FUNCTION_BLOCK FB_TimeSwitch_V2
VAR_INPUT
	b_Enable: BOOL;
	b_StatusOn: BOOL;
	structSystemTime: timestruct;
	byte_MoFr_Open_Hour: BYTE;
	byte_MoFr_Open_Minute: BYTE;
	byte_MoFr_Close_Hour: BYTE;
	byte_MoFr_Close_Minute: BYTE;
	byte_Sa_Open_Hour: BYTE;
	byte_Sa_Open_Minute: BYTE;
	byte_Sa_Close_Hour: BYTE;
	byte_Sa_Close_Minute: BYTE;	
	byte_So_Open_Hour: BYTE;
	byte_So_Open_Minute: BYTE;
	byte_So_Close_Hour: BYTE;
	byte_So_Close_Minute: BYTE;
	real_Offset_Start: REAL;
	real_Offset_Stop: REAL;	
	b_On_Manual: BOOL;
	b_Off_Manual: BOOL;
END_VAR
VAR_OUTPUT
	b_Output_On: BOOL;
	b_Error: BOOL;
END_VAR
VAR
	TON_0: ton;
	byte_Day :BYTE;		// 0: Sunday, 1: Monday,....
	time_now             		: TIME;
	time_MoFr_Open             	: TIME;
	time_MoFr_Close             : TIME;
	time_Sa_Open             	: TIME;
	time_Sa_Close             	: TIME;
	time_So_Open             	: TIME;
	time_So_Close             	: TIME;
	

	RS_0: rs;
	R_TRIG_0: r_trig;
	R_TRIG_1: r_trig;
	dt_Test: DATE_AND_TIME;
	tod_test: TIME_OF_DAY;
	time_temp: TIME;
	time_Start_MoFr_Calc: TIME;
	time_Stop_MoFr_Calc: TIME;
	time_Start_Sa_Calc: TIME;
	time_Stop_Sa_Calc: TIME;
	time_Start_So_Calc: TIME;
	time_Stop_So_Calc: TIME;
	
	FB_WeeklyTimeSwitch_MoFr: FB_WeeklyTimeSwitch;
	FB_WeeklyTimeSwitch_Sa: FB_WeeklyTimeSwitch;
	FB_WeeklyTimeSwitch_So: FB_WeeklyTimeSwitch;
	RS_manu: rs;
	b_Auto_on: BOOL;

	R_TRIG_2: r_trig;
	R_TRIG_3: r_trig;
	F_TRIG_0: f_trig;
	R_TRIG_4: r_trig;
	R_TRIG_FirstCycle: r_trig;
	time_Zero             	: TIME;
	
END_VAR
VAR // added by the converter: edge detectors and wires of the graphical bodies
    _w1 : DATE_AND_TIME;
    _w2 : TIME_OF_DAY;
    _w3 : BOOL;
END_VAR

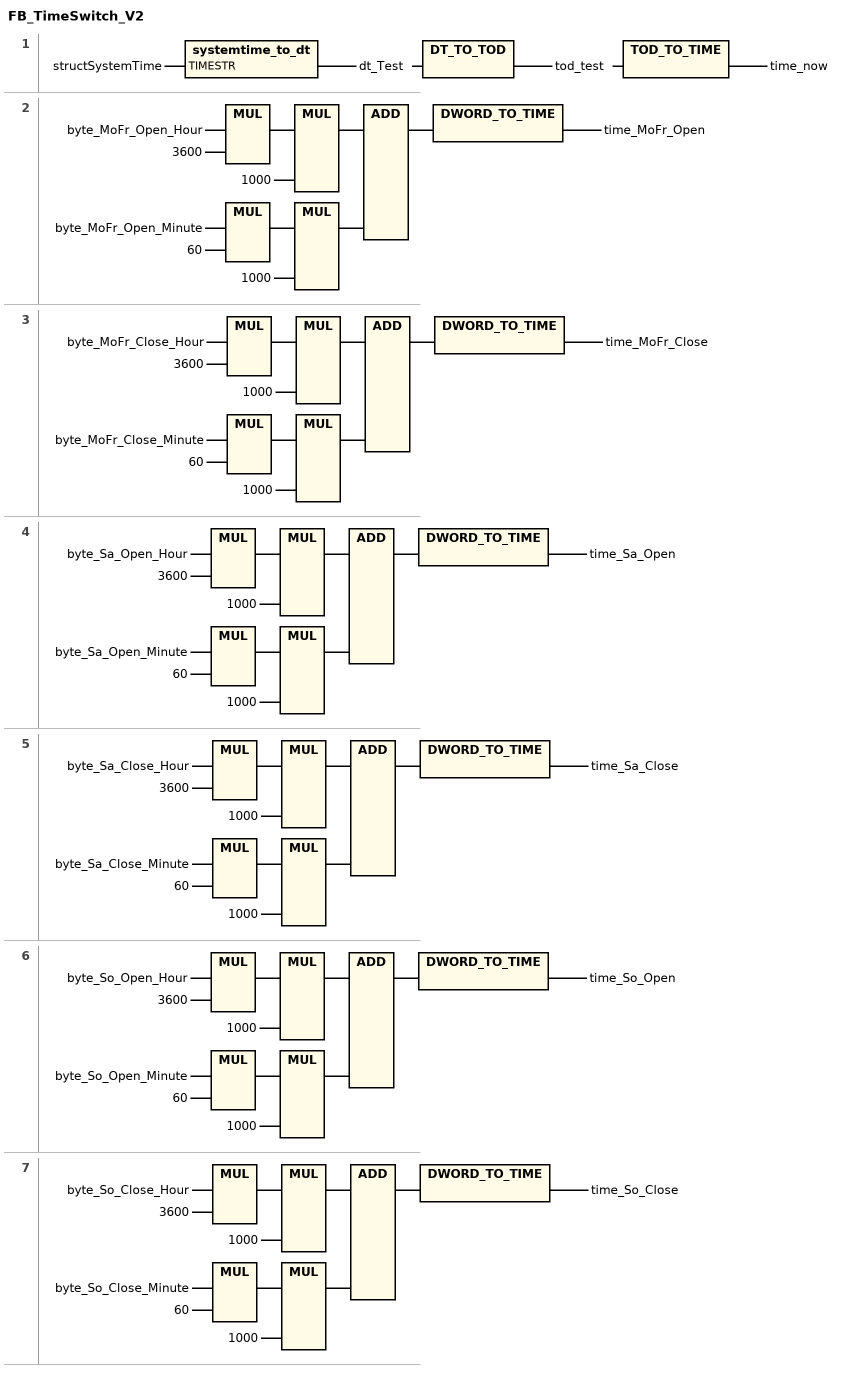
// NETWORK 1
_w1 := systemtime_to_dt(TIMESTR := structSystemTime);
dt_Test := _w1;
_w2 := DT_TO_TOD(_w1);
tod_test := _w2;
time_now := TOD_TO_TIME(_w2);

// NETWORK 2
time_MoFr_Open := DWORD_TO_TIME((byte_MoFr_Open_Hour * 3600) * 1000 + (byte_MoFr_Open_Minute * 60) * 1000);

// NETWORK 3
time_MoFr_Close := DWORD_TO_TIME((byte_MoFr_Close_Hour * 3600) * 1000 + (byte_MoFr_Close_Minute * 60) * 1000);

// NETWORK 4
time_Sa_Open := DWORD_TO_TIME((byte_Sa_Open_Hour * 3600) * 1000 + (byte_Sa_Open_Minute * 60) * 1000);

// NETWORK 5
time_Sa_Close := DWORD_TO_TIME((byte_Sa_Close_Hour * 3600) * 1000 + (byte_Sa_Close_Minute * 60) * 1000);

// NETWORK 6
time_So_Open := DWORD_TO_TIME((byte_So_Open_Hour * 3600) * 1000 + (byte_So_Open_Minute * 60) * 1000);

// NETWORK 7
time_So_Close := DWORD_TO_TIME((byte_So_Close_Hour * 3600) * 1000 + (byte_So_Close_Minute * 60) * 1000);

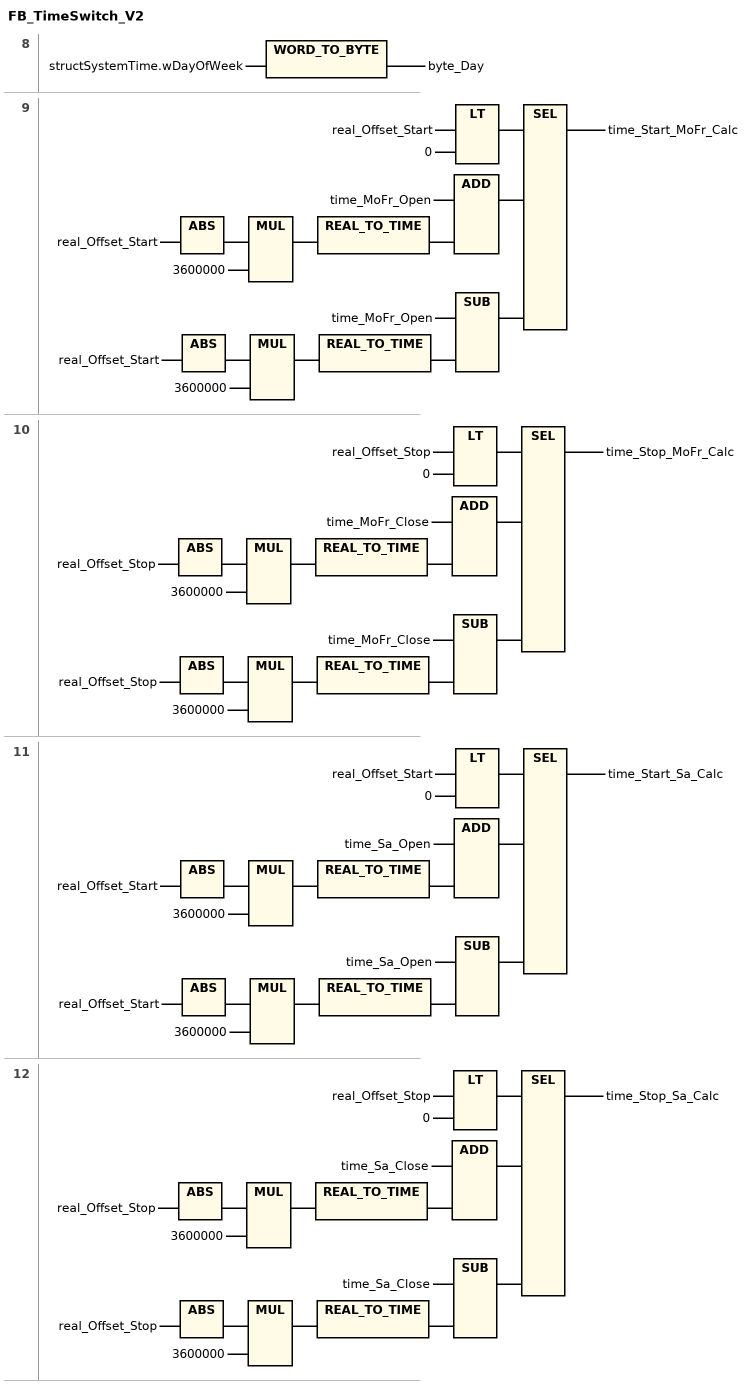
// NETWORK 8
byte_Day := WORD_TO_BYTE(structSystemTime.wDayOfWeek);

// NETWORK 9
time_Start_MoFr_Calc := SEL(real_Offset_Start < 0, time_MoFr_Open + REAL_TO_TIME(ABS(real_Offset_Start) * 3600000), time_MoFr_Open - REAL_TO_TIME(ABS(real_Offset_Start) * 3600000));

// NETWORK 10
time_Stop_MoFr_Calc := SEL(real_Offset_Stop < 0, time_MoFr_Close + REAL_TO_TIME(ABS(real_Offset_Stop) * 3600000), time_MoFr_Close - REAL_TO_TIME(ABS(real_Offset_Stop) * 3600000));

// NETWORK 11
time_Start_Sa_Calc := SEL(real_Offset_Start < 0, time_Sa_Open + REAL_TO_TIME(ABS(real_Offset_Start) * 3600000), time_Sa_Open - REAL_TO_TIME(ABS(real_Offset_Start) * 3600000));

// NETWORK 12
time_Stop_Sa_Calc := SEL(real_Offset_Stop < 0, time_Sa_Close + REAL_TO_TIME(ABS(real_Offset_Stop) * 3600000), time_Sa_Close - REAL_TO_TIME(ABS(real_Offset_Stop) * 3600000));

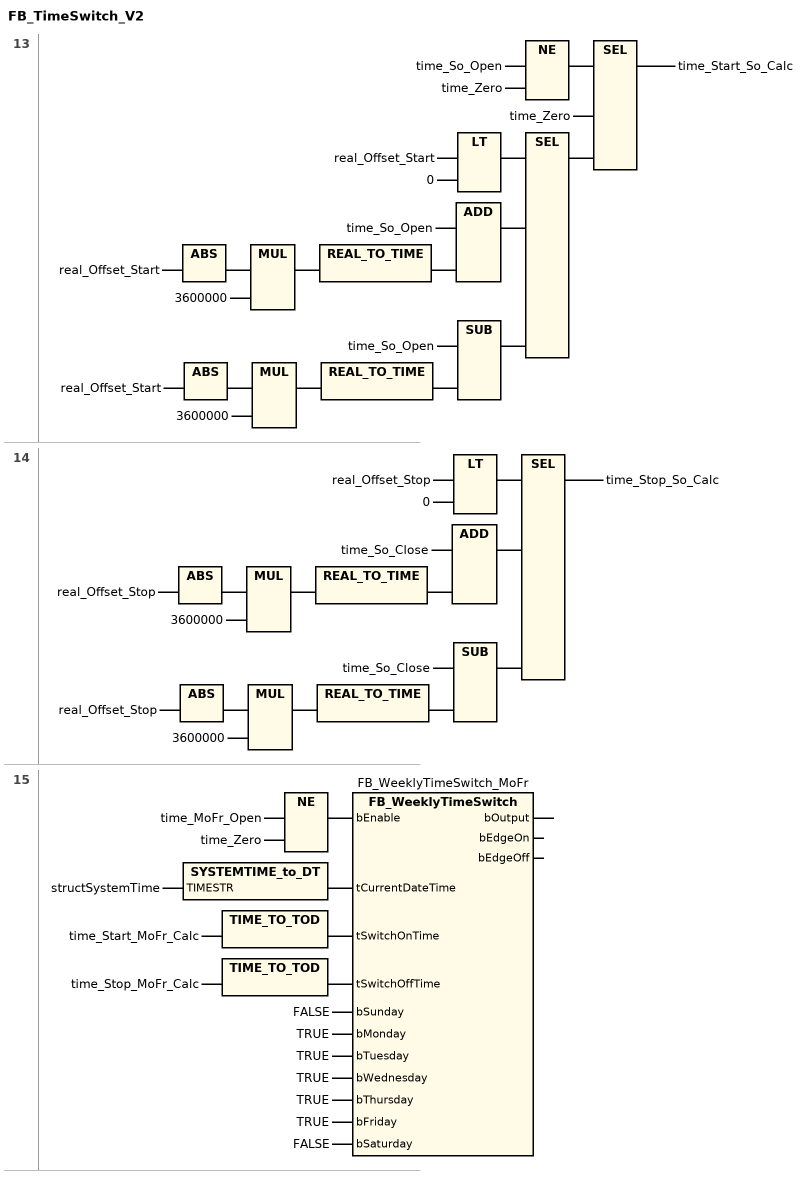
// NETWORK 13
time_Start_So_Calc := SEL(time_So_Open <> time_Zero, time_Zero, SEL(real_Offset_Start < 0, time_So_Open + REAL_TO_TIME(ABS(real_Offset_Start) * 3600000), time_So_Open - REAL_TO_TIME(ABS(real_Offset_Start) * 3600000)));

// NETWORK 14
time_Stop_So_Calc := SEL(real_Offset_Stop < 0, time_So_Close + REAL_TO_TIME(ABS(real_Offset_Stop) * 3600000), time_So_Close - REAL_TO_TIME(ABS(real_Offset_Stop) * 3600000));

// NETWORK 15
FB_WeeklyTimeSwitch_MoFr(
    bEnable := time_MoFr_Open <> time_Zero,
    tCurrentDateTime := SYSTEMTIME_to_DT(TIMESTR := structSystemTime),
    tSwitchOnTime := TIME_TO_TOD(time_Start_MoFr_Calc),
    tSwitchOffTime := TIME_TO_TOD(time_Stop_MoFr_Calc),
    bSunday := FALSE,
    bMonday := TRUE,
    bTuesday := TRUE,
    bWednesday := TRUE,
    bThursday := TRUE,
    bFriday := TRUE,
    bSaturday := FALSE); // FB_WeeklyTimeSwitch

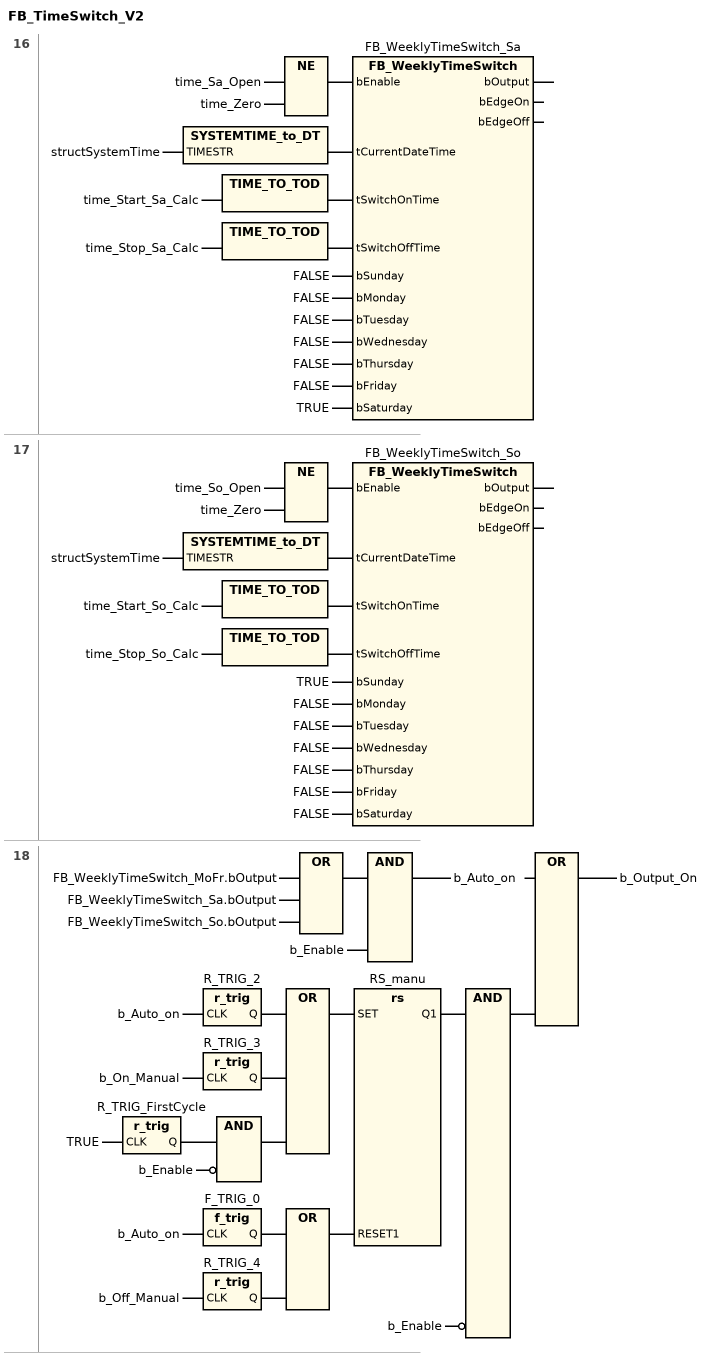
// NETWORK 16
FB_WeeklyTimeSwitch_Sa(
    bEnable := time_Sa_Open <> time_Zero,
    tCurrentDateTime := SYSTEMTIME_to_DT(TIMESTR := structSystemTime),
    tSwitchOnTime := TIME_TO_TOD(time_Start_Sa_Calc),
    tSwitchOffTime := TIME_TO_TOD(time_Stop_Sa_Calc),
    bSunday := FALSE,
    bMonday := FALSE,
    bTuesday := FALSE,
    bWednesday := FALSE,
    bThursday := FALSE,
    bFriday := FALSE,
    bSaturday := TRUE); // FB_WeeklyTimeSwitch

// NETWORK 17
FB_WeeklyTimeSwitch_So(
    bEnable := time_So_Open <> time_Zero,
    tCurrentDateTime := SYSTEMTIME_to_DT(TIMESTR := structSystemTime),
    tSwitchOnTime := TIME_TO_TOD(time_Start_So_Calc),
    tSwitchOffTime := TIME_TO_TOD(time_Stop_So_Calc),
    bSunday := TRUE,
    bMonday := FALSE,
    bTuesday := FALSE,
    bWednesday := FALSE,
    bThursday := FALSE,
    bFriday := FALSE,
    bSaturday := FALSE); // FB_WeeklyTimeSwitch

// NETWORK 18
_w3 := (FB_WeeklyTimeSwitch_MoFr.bOutput OR FB_WeeklyTimeSwitch_Sa.bOutput OR FB_WeeklyTimeSwitch_So.bOutput) AND b_Enable;
b_Auto_on := _w3;
R_TRIG_2(CLK := b_Auto_on); // r_trig
R_TRIG_3(CLK := b_On_Manual); // r_trig
R_TRIG_FirstCycle(CLK := TRUE); // r_trig
F_TRIG_0(CLK := b_Auto_on); // f_trig
R_TRIG_4(CLK := b_Off_Manual); // r_trig
RS_manu(SET := R_TRIG_2.Q OR R_TRIG_3.Q OR R_TRIG_FirstCycle.Q AND NOT b_Enable, RESET1 := F_TRIG_0.Q OR R_TRIG_4.Q); // rs
b_Output_On := _w3 OR RS_manu.Q1 AND NOT b_Enable;

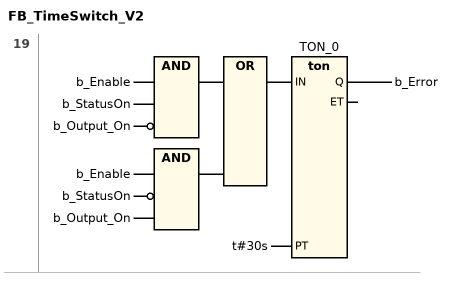
// NETWORK 19
TON_0(IN := b_Enable AND b_StatusOn AND NOT b_Output_On OR b_Enable AND NOT b_StatusOn AND b_Output_On, PT := t#30s); // ton
b_Error := TON_0.Q;

END_FUNCTION_BLOCK

(* stored: Version 1.1.0.1, ProductVersion 3.1.4024.11
   POU FB_TimeSwitch_V2: Id {cc23047c-7723-456a-a19f-31e83741e9a1}, SpecialFunc None *)
